KUKA KRL program: Station3.src, Station3.dat

--- Station3.src ---
&ACCESS RV
DEF Station3 (lnTargetSt :IN)
   INT lnTargetSt

   IF(gnActSt <> lnTargetSt) THEN
      MoveTo (gnActSt,lnTargetSt)
   ENDIF

   REPEAT
   UNTIL gnActSt ==lnTargetSt

   CONTINUE
   IF NOT (gnActSt == lnTargetSt) THEN
      LOOP
         HALT
      ENDLOOP
   ENDIF
    WAIT SEC 0
   ;; TO DO
   St3_Job1(lnTargetSt, gnLastToolNr)
   gbProbeCalibrated = TRUE


   CONTINUE
   IF gbRecoveryNeeded  THEN
      HALT
      IF NOT RecoverFromWorkSt(lnTargetSt)  THEN
         boRobotUnknowPos =  TRUE
         LOOP
            HALT
         ENDLOOP
      ENDIF
   ENDIF
END

--- Station3.dat ---
&ACCESS RV
DEFDAT  Station3 PUBLIC

ENDDAT
